// TIA Portal V17 export
// export: Created 2022-07-20T07:01:32.1606698Z, ExportSetting WithDefaults, DisplayName Totally Integrated Automation Portal, DisplayVersion V17, DisplayName TIA Portal Openness, DisplayVersion V17, DisplayName TIA Portal Version Control Interface, DisplayVersion V17, DisplayName SINAMICS Startdrive Advanced, DisplayVersion V17, DisplayName SINAMICS Startdrive G130, G150, S120, S150, SINAMICS MV, S210, DisplayVersion V17, DisplayName SINAMICS Startdrive G110M, G120, G120C, G120D, G120P, G115D, DisplayVersion V17, DisplayName STEP 7 Professional, DisplayVersion V17, DisplayName STEP 7 Safety, DisplayVersion V17, DisplayName WinCC Advanced, DisplayVersion V17
FUNCTION_BLOCK "FB10342_WebGuide"   // FB10342, LAD
TITLE = FB10342_WebGuide
{ S7_Optimized_Access := 'TRUE' }
VERSION : 0.1
// stored: AutoNumber false, IsIECCheckEnabled false, IsRetainMemResEnabled false, MemoryReserve 100, SetENOAutomatically false, UDAEnableTagReadback false
   VAR_INPUT
      RequestAcknowledge : Bool;
   END_VAR
   VAR_OUTPUT
      ActiveWebGuide : Bool;
      WebGuideActivated : Bool;
      WebGuideInError : Bool;
   END_VAR
   VAR_IN_OUT
      RequestActiveWebGuide : Bool;
   END_VAR
   VAR
      R_TRIG_RequestActiveWebGuide : R_TRIG;
      F_TRIG_RequestActiveWebGuide { S7_SetPoint := 'True'} : F_TRIG;
      TON_WebGuideActivated { S7_SetPoint := 'True'} : TON_TIME;
      TON_WebGuideNotActivated { S7_SetPoint := 'True'} : TON_TIME;
      TON_WebGuideInError { S7_SetPoint := 'True'} : TON_TIME;
   END_VAR
BEGIN

REGION Network 1 (SCL): First Scan
   IF "FirstScan" THEN
       #ActiveWebGuide := FALSE;
   END_IF;
END_REGION

REGION Network 2 (SCL): Edge Signals & Timers
   REGION EDGE SIGNALS
       #R_TRIG_RequestActiveWebGuide(CLK := #RequestActiveWebGuide);
       #F_TRIG_RequestActiveWebGuide(CLK := #RequestActiveWebGuide);
   END_REGION

   REGION TIMERS
       #TON_WebGuideActivated(IN := #ActiveWebGuide,
                             PT := T#2s);
      #TON_WebGuideNotActivated(IN := NOT (#ActiveWebGuide),
                                PT := T#2s);
       #TON_WebGuideInError(IN := #RequestActiveWebGuide AND NOT (#ActiveWebGuide)
                            OR #RequestActiveWebGuide AND NOT (#WebGuideActivated)
                            OR NOT (#RequestActiveWebGuide) AND #ActiveWebGuide
                            OR NOT (#RequestActiveWebGuide) AND #WebGuideActivated, PT := T#10s);
   END_REGION
END_REGION

REGION Network 3 (SCL): WebGuide Management
   IF #R_TRIG_RequestActiveWebGuide.Q THEN
       #ActiveWebGuide := TRUE;
   ELSIF #F_TRIG_RequestActiveWebGuide.Q THEN
       #ActiveWebGuide := FALSE;
   END_IF;
END_REGION

REGION Network 4 (SCL): States
   IF #TON_WebGuideActivated.Q THEN
       #WebGuideActivated := TRUE;
   ELSIF #TON_WebGuideNotActivated.Q THEN
       #WebGuideActivated := FALSE;
   END_IF;

   IF #TON_WebGuideInError.Q THEN
       #WebGuideInError := TRUE;
   ELSIF #RequestAcknowledge THEN
       #WebGuideInError := FALSE;
   END_IF;
END_REGION
END_FUNCTION_BLOCK
